FUNCTION_BLOCK FB_MotionRef
VAR_INPUT
	
END_VAR
VAR_OUTPUT
	
END_VAR
VAR
	
END_VAR

END_FUNCTION_BLOCK

(* stored: Version 1.1.0.1
   POU FB_MotionRef: Id {c8c75e4f-5790-4c91-ac23-d3af2bcb69cb}, SpecialFunc None *)
